(* IEC 61131-3 sources: AutoCam_Corralon/plc/src, 3 files *)

(* ---- alarms.st ---- *)
FUNCTION_BLOCK FB_Alarms
VAR_INPUT
    LevelSensorOK : BOOL;
    LevelLitres   : REAL;
    MinimumLevel  : REAL;
END_VAR

VAR_OUTPUT
    AlarmSensor   : BOOL;
    AlarmLowLevel : BOOL;
    AlarmGeneral  : BOOL;
END_VAR

AlarmSensor   := NOT LevelSensorOK;
AlarmLowLevel := LevelSensorOK AND (LevelLitres <= MinimumLevel);
AlarmGeneral  := AlarmSensor OR AlarmLowLevel;

END_FUNCTION_BLOCK

(* ---- irrigation.st ---- *)
FUNCTION_BLOCK FB_IrrigationLine
VAR_INPUT
    Command      : BOOL;
    SystemEnable : BOOL;
    AlarmGeneral : BOOL;
END_VAR

VAR_OUTPUT
    Valve : BOOL;
END_VAR

Valve :=
    Command
    AND SystemEnable
    AND NOT AlarmGeneral;

END_FUNCTION_BLOCK

(* ---- pump_control.st ---- *)
FUNCTION_BLOCK FB_PumpControl
VAR_INPUT
    Command      : BOOL;
    SensorOK     : BOOL;
    LevelLitres  : REAL;
    MinimumLevel : REAL;
    AlarmGeneral : BOOL;
END_VAR

VAR_OUTPUT
    Permission : BOOL;
    Pump       : BOOL;
END_VAR

Permission :=
    SensorOK
    AND (LevelLitres > MinimumLevel)
    AND NOT AlarmGeneral;

Pump := Command AND Permission;

END_FUNCTION_BLOCK
